PROGRAM Axis_11_Function_Blocks
VAR
END_VAR

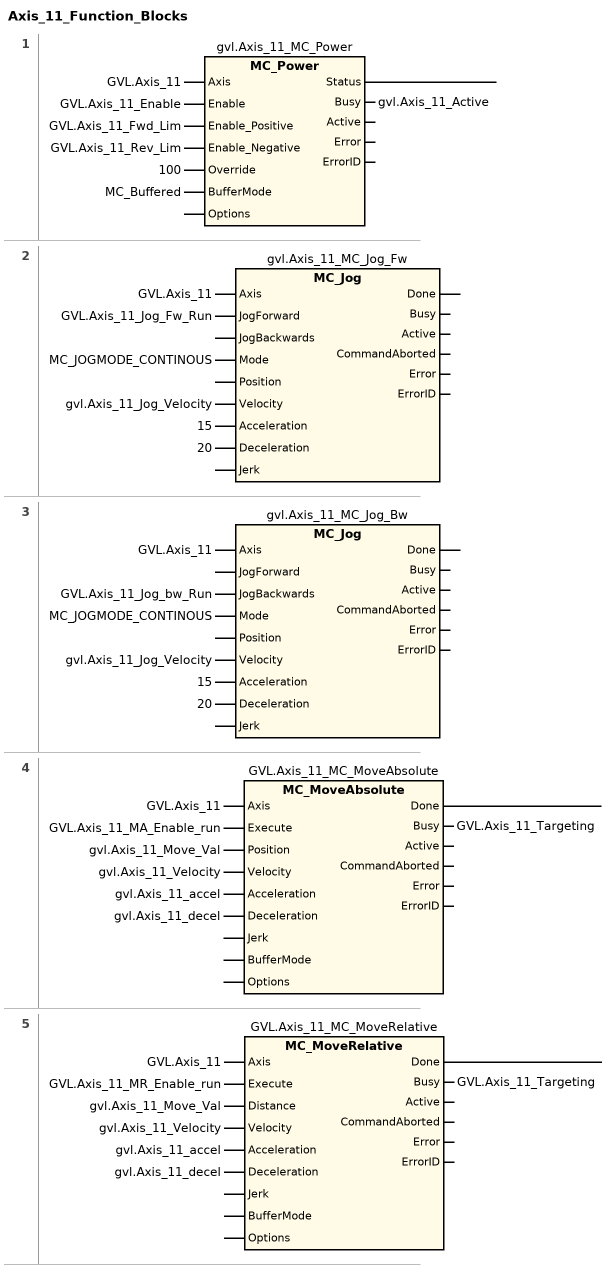
// NETWORK 1
gvl.Axis_11_MC_Power(
    Axis := GVL.Axis_11,
    Enable := GVL.Axis_11_Enable,
    Enable_Positive := GVL.Axis_11_Fwd_Lim,
    Enable_Negative := GVL.Axis_11_Rev_Lim,
    Override := 100,
    BufferMode := MC_Buffered,
    Busy => gvl.Axis_11_Active); // MC_Power

// NETWORK 2
gvl.Axis_11_MC_Jog_Fw(
    Axis := GVL.Axis_11,
    JogForward := GVL.Axis_11_Jog_Fw_Run,
    Mode := MC_JOGMODE_CONTINOUS,
    Velocity := gvl.Axis_11_Jog_Velocity,
    Acceleration := 15,
    Deceleration := 20); // MC_Jog

// NETWORK 3
gvl.Axis_11_MC_Jog_Bw(
    Axis := GVL.Axis_11,
    JogBackwards := GVL.Axis_11_Jog_bw_Run,
    Mode := MC_JOGMODE_CONTINOUS,
    Velocity := gvl.Axis_11_Jog_Velocity,
    Acceleration := 15,
    Deceleration := 20); // MC_Jog

// NETWORK 4
GVL.Axis_11_MC_MoveAbsolute(
    Axis := GVL.Axis_11,
    Execute := GVL.Axis_11_MA_Enable_run,
    Position := gvl.Axis_11_Move_Val,
    Velocity := gvl.Axis_11_Velocity,
    Acceleration := gvl.Axis_11_accel,
    Deceleration := gvl.Axis_11_decel,
    Busy => GVL.Axis_11_Targeting); // MC_MoveAbsolute

// NETWORK 5
GVL.Axis_11_MC_MoveRelative(
    Axis := GVL.Axis_11,
    Execute := GVL.Axis_11_MR_Enable_run,
    Distance := gvl.Axis_11_Move_Val,
    Velocity := gvl.Axis_11_Velocity,
    Acceleration := gvl.Axis_11_accel,
    Deceleration := gvl.Axis_11_decel,
    Busy => GVL.Axis_11_Targeting); // MC_MoveRelative

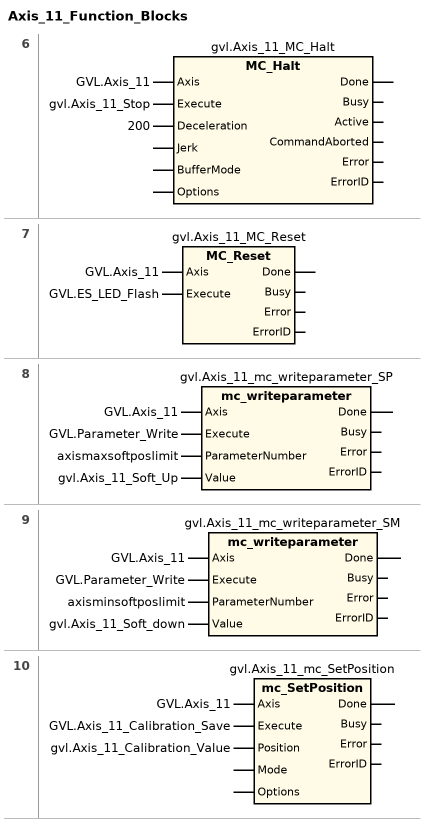
// NETWORK 6
gvl.Axis_11_MC_Halt(Axis := GVL.Axis_11, Execute := gvl.Axis_11_Stop, Deceleration := 200); // MC_Halt

// NETWORK 7
gvl.Axis_11_MC_Reset(Axis := GVL.Axis_11, Execute := GVL.ES_LED_Flash); // MC_Reset

// NETWORK 8
gvl.Axis_11_mc_writeparameter_SP(
    Axis := GVL.Axis_11,
    Execute := GVL.Parameter_Write,
    ParameterNumber := axismaxsoftposlimit,
    Value := gvl.Axis_11_Soft_Up); // mc_writeparameter

// NETWORK 9
gvl.Axis_11_mc_writeparameter_SM(
    Axis := GVL.Axis_11,
    Execute := GVL.Parameter_Write,
    ParameterNumber := axisminsoftposlimit,
    Value := gvl.Axis_11_Soft_down); // mc_writeparameter

// NETWORK 10
gvl.Axis_11_mc_SetPosition(
    Axis := GVL.Axis_11,
    Execute := GVL.Axis_11_Calibration_Save,
    Position := gvl.Axis_11_Calibration_Value); // mc_SetPosition

END_PROGRAM

(* stored: Version 1.1.0.1, ProductVersion 3.1.4022.12
   POU Axis_11_Function_Blocks: Id {f1bed9e8-6a49-4307-a1b4-d4a5090a9a41}, SpecialFunc None *)
